Staubli VAL3: iPilatusPos.pgx

public program iPilatusPos(num& nNum[] (dimensions=1))
begin
  nNum=dioGet(iPilatusPos)
end
